FUNCTION_BLOCK NOT_42C76073DCEB1A7A (* Logical NOT *)
  (* Standard: 61499-2 *)
  (* Version 1.0, 24.09.2008, marumil, nxtControl GmbH, Initial Version *)
  PACKAGE UAO.Hackathon;
  (* Compiler Cpp *)
  {SET_ATTRIBUTE(Runtime.FBType.ImplementingType, Runtime.Standard#DYNGEN_NOT)}
  {SET_ATTRIBUTE(Configuration.GenericFBType.InterfaceParams, Runtime.Standard#CNT:=1;OUT${CNT$}:BOOL)}
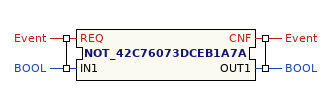
  EVENT_INPUT
    REQ WITH IN1; (* Normal Execution Request *)
  END_EVENT
  EVENT_OUTPUT
    CNF WITH OUT1; (* Execution Confirmation *)
  END_EVENT
  VAR_INPUT
    IN1 : BOOL; (* Argument *)
  END_VAR
  VAR_OUTPUT
    OUT1 : BOOL; (* Result: NOT INn *)
  END_VAR
  EC_STATES
    START;
  END_STATES
END_FUNCTION_BLOCK
